TYPE ST_Loadbank_params :
STRUCT
	b_Enable					: BOOL;
	r_PowerRating				: REAL; // kW
	r_PowerStepSize				: REAL; // kW
END_STRUCT
END_TYPE

(* stored: Version 1.1.0.1, ProductVersion 3.1.4026.18
   DUT ST_Loadbank_params: Id {a08f514c-9524-4cb3-99ec-d82215ccfa88} *)
